FUNCTION ScaleSpeed : UINT
VAR_INPUT
	iSpeed : UINT;
	SpeedMatrix	: ARRAY[0..Constants.speedMatrixSize] OF FfuSpeed;
END_VAR
VAR
	i : UINT;
	found	: BOOL := FALSE;
END_VAR

FOR i:= 1 TO Constants.speedMatrixSize DO
	IF (SpeedMatrix[i].NonScaledSpeedValue = iSpeed) THEN
		ScaleSpeed := SpeedMatrix[i].ScaledSpeedValue;
		found := TRUE;
	EXIT;
	END_IF
END_FOR

IF NOT found THEN
	ScaleSpeed := 0;
END_IF

END_FUNCTION

(* stored: Version 1.1.0.1, ProductVersion 3.1.4024.12
   POU ScaleSpeed: Id {f2fb93aa-4683-43c7-87a6-d19d37e1f8b5}, SpecialFunc None *)
